(* Logix 5000 project; controller TWO_SRC_TEST vendor 1 type 14 code 54 rev 19.11; software revision 19.01 *)
// Two sources are connected to the same bus and power is shared between the two using a voltage droop controller.

TASK MainTask (continuous, watchdog 500 ms) : MainProgram

MODULES
   Local : vendor 1 type 14 code 54 (ICP 0, rev 19.11)
      CurrentMeasurement : 1756-IF8 (ICP 2, rev 1.1, Input RPI 100 ms)
      VoltageSetpoints : 1756-OF4 (ICP 1, rev 1.1, Output RPI 12 ms)
END_MODULES

VAR_GLOBAL   (* controller tags *)
   SOURCE_1_Current : ALIAS FOR Local:2:I.Ch0Data;
   SOURCE_2_Current : ALIAS FOR Local:2:I.Ch1Data;
END_VAR

PROGRAM MainProgram   (* main routine MainRoutine *)
VAR
   CURRENT_SCALING_FACTOR : REAL;
   MeasArray : COUNTER;
   MeasCount : COUNTER;
   MeasCounter : COUNTER;
   MeasTimer : TIMER := (PRE := 10);
   SOURCE_1_CurrentBuffer : REAL;
   SOURCE_1_DeltaV : REAL;
   SOURCE_1_DroopCoefficient : REAL;
   SOURCE_1_FullLoadCurrent : REAL;
   SOURCE_1_FullLoadVoltage : REAL;
   SOURCE_1_NoLoadVoltage : REAL;
   SOURCE_1_OutputVoltage : REAL;
   SOURCE_1_VoltageAdjustment : REAL;
END_VAR

ROUTINE MainRoutine   (* ladder *)
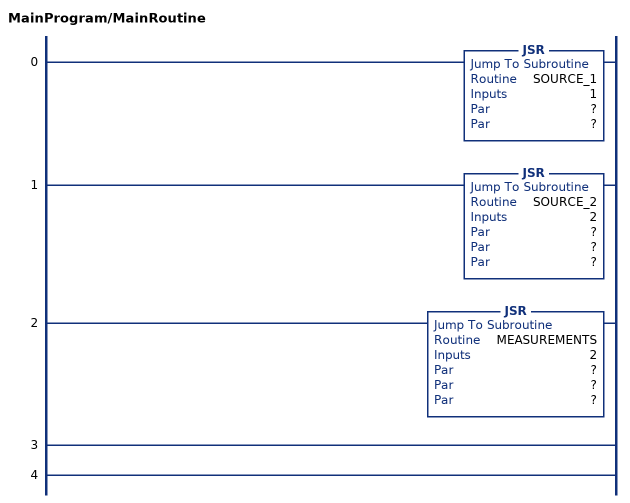
   0: JSR(SOURCE_1,1,?,?);
   1: JSR(SOURCE_2,2,?,?,?);
   2: JSR(MEASUREMENTS,2,?,?,?);
   3: ;
   4: ;
END_ROUTINE

ROUTINE MEASUREMENTS   (* ladder *)
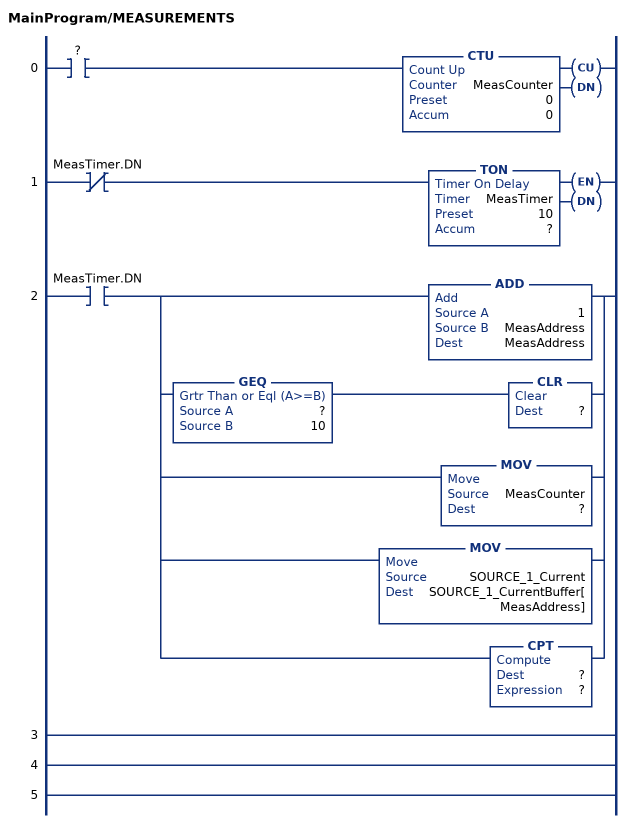
   0: XIC(?)CTU(MeasCounter,0,0);
   1: XIO(MeasTimer.DN)TON(MeasTimer,?,?);
   2: XIC(MeasTimer.DN)[ADD(1,MeasAddress,MeasAddress) ,GEQ(?,10) CLR(?) ,MOV(MeasCounter,?) ,MOV(SOURCE_1_Current,SOURCE_1_CurrentBuffer[MeasAddress]) ,CPT(?,?) ];
   3: ;
   4: ;
   5: ;
END_ROUTINE

ROUTINE SOURCE_1   (* ladder *)
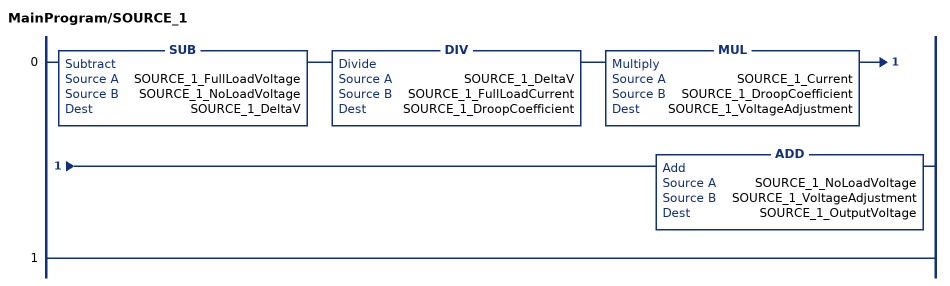
   0: SUB(SOURCE_1_FullLoadVoltage,SOURCE_1_NoLoadVoltage,SOURCE_1_DeltaV)DIV(SOURCE_1_DeltaV,SOURCE_1_FullLoadCurrent,SOURCE_1_DroopCoefficient)MUL(SOURCE_1_Current,SOURCE_1_DroopCoefficient,SOURCE_1_VoltageAdjustment)ADD(SOURCE_1_NoLoadVoltage,SOURCE_1_VoltageAdjustment,SOURCE_1_OutputVoltage);
   1: ;
END_ROUTINE
END_PROGRAM
